PROGRAM MAIN
VAR
	nCounter			:INT;
	sText				:STRING;
	bFlag				:BOOL;
	bQuit				:BOOL;
	
	step				:INT;
END_VAR


IF bFlag THEN
	step := step + 1;
END_IF

IF step > 20 THEN
	//bFlag := FALSE;	// limit to 1 msg as a test
	nCounter := nCounter + 1;
	IF nCounter > 32000 THEN nCounter := 1; END_IF
	
	sMsg_SCP_Event(100,
		nCounter, '',
		0, '',
		0, '',
		0, '',
		0, '',
		0, '',
		0, '');

	step := 0;
END_IF




P800_Core_Messaging();

IF bQuit THEN
	bQuit := FALSE;
	vMessages.Msgs_SCP.Pending := 'quit';
END_IF

END_PROGRAM

(* stored: Version 1.1.0.1, ProductVersion 3.1.4024.9
   POU MAIN: Id {634c16e4-9cae-4701-9e3b-d0bbcebd34bb}, SpecialFunc None *)
